FUNCTION_BLOCK FB_Winter EXTENDS FB_SeasonBase
VAR
END_VAR

METHOD ChangeToWinterTyres
VAR_INPUT
END_VAR
THIS^._nTyresType := 0;
Tc2_System.ADSLOGSTR(msgCtrlMask := THIS^._nLogLevel,
                     msgFmtStr := 'Changed to winter tyres',
                     strArg := '');
END_METHOD

METHOD FB_init : BOOL
VAR_INPUT
    bInitRetains:           BOOL; // if TRUE, the retain variables are initialized (warm start / cold start)
    bInCopyCode:            BOOL;  // if TRUE, the instance afterwards gets moved into the copy code (online change)
    ipStateMachine:         I_StateMachine;
    ipParentObject:         I_Object;
END_VAR
THIS^._eState := E_Season.Winter;
END_METHOD

METHOD  NextSeason
VAR_INPUT
END_VAR
THIS^.ipStateMachine.SetState(THIS^.ipSeasonCtrl.StateSpring);
END_METHOD

METHOD OnEntry
VAR_INPUT
END_VAR
SUPER^.OnEntry();
THIS^._bWindBlowing     := FALSE;
THIS^._bRaining         := FALSE;
THIS^._bSunShining      := FALSE;
THIS^._bSnowing         := TRUE;
THIS^._nLeavesState     := 0;
END_METHOD

END_FUNCTION_BLOCK

(* stored: Version 1.1.0.1, ProductVersion 3.1.4024.12
   POU FB_Winter: Id {dd31ff79-7608-4329-a882-f2a214963310}, SpecialFunc None
   Method ChangeToWinterTyres: Id {c501c20b-7321-4fa1-a0b0-2cdf840d0f58}
   Method FB_init: Id {c1eab856-cdeb-4166-80be-5147b9676904}
   Method NextSeason: Id {02e5b18e-46a5-400f-9dbd-20c607af148e}
   Method OnEntry: Id {1bf1e8f4-4927-4afd-9926-3fdb068689d2} *)
